(*
SPDX-FileCopyrightText: © 2026 Oleksandr Tiutyk <trofimich@gmail.com>
SPDX-License-Identifier: MIT
License: https://opensource.org/license/mit
*)

TYPE JSON_DOCUMENT : STRING(25000); END_TYPE

(* stored: Version 1.1.0.1
   DUT JSON_DOCUMENT: Id {1c584fbf-bc67-4669-8e1b-884fc72f5a93} *)
